FUNCTION_BLOCK FB_ActuatorLinear 

VAR	
	axis: 				AXIS_REF;
	power: 				MC_Power;
	powerOutputs: 		ST_McOutputs;
	moveAbs: 			MC_MoveAbsolute;
	moveAbsOutputs: 	ST_McOutputs;
	reset: 				MC_Reset;
	resetOut: 			ST_McOutputs;
	home:				MC_Home;
	
	
	sID: STRING;
	sDescr: STRING;
	
	
	nLead: UINT := 5;  			// mm per 360deg  - NOT EFFECTIVE YET BECAUSE PITCH IS CURRENTLY HANDLED IN THE AXIS CONFIG
	nStroke: UINT := 100;  		// length of travel
	nHomeOffset: UINT := 0; 	// offset distance from hard-stop for home
	nMaxVel: UINT := 300; 		// mm/s
	nPercentMove: LREAL := 100; 	// % of the full extent of movement (starting from position 0)
	
	eSMState: (INIT, ENABLE, WAIT, FWD_TRIG, FWD, REV_TRIG, REV, ERROR, RESET, HOMING, HOME) := INIT;
	
	fbTONDelay: TON := (PT := T#5S);
	bFirstRun: BOOL := TRUE;
	

	
END_VAR

ActMove();
ActPower();
ActReset();
fbTONDelay();


CASE eSMState OF
	
	INIT:

		IF bFirstRun THEN
			fbTONDelay.IN := TRUE;
			bFirstRun := FALSE;
		END_IF
		
		moveAbs.Execute := FALSE;
		moveAbs.Execute := FALSE;
		reset.Execute := FALSE;
		
		
		IF fbTONDelay.Q THEN
			eSMState := ENABLE;
			fbTONDelay.IN := FALSE;	
			bFirstRun := TRUE;
		END_IF
		
		
		
		
	ENABLE:
	
		IF bFirstRun THEN
			fbTONDelay.IN := TRUE;
			bFirstRun := FALSE;
		END_IF
	
		
		power.Enable := TRUE;
		power.Enable_Positive := TRUE;
		power.Enable_Negative := TRUE;
		
		
		IF power.Status THEN
			eSMState := WAIT;
			fbTONDelay.IN := FALSE;	
			bFirstRun := TRUE;
		(* ELSIF power.Error AND fbTONDelay.Q THEN
			eSMState := ERROR;
			fbTONDelay.IN := FALSE;
			bFirstRun := TRUE; *)
		END_IF
		
	WAIT:
		// Handle eStateTarget command requests here 
		//IF eStateTarget := E_DeviceState.
		
	
	HOMING:
		
		
	FWD_TRIG:
			
			moveAbs.Position := - nStroke * (nPercentMove / 100);		(* mm *)
			moveAbs.Velocity := nMaxVel/2;		(* mm/s *)
			moveAbs.BufferMode := MC_Buffered;  
			moveAbs.Execute := TRUE;
			
			IF moveAbs.Active THEN
				moveAbs.Execute := FALSE;
				fbTONDelay.IN := FALSE;
				eSMState := FWD;
				bFirstRun := TRUE;
			ELSIF moveAbs.CommandAborted OR moveAbs.Error THEN
				eSMState := ERROR;
				bFirstRun := TRUE;
				moveAbs.Execute := FALSE;
			END_IF
				
	FWD:
			eSMState := INIT;
			//eState := FWD;
			
			
			
			
	REV_TRIG:
	
			moveAbs.Position := - (0 + nHomeOffset)  * (nPercentMove / 100);		(* mm *)
			moveAbs.Velocity := nMaxVel/2;										(* mm/s *)
			moveAbs.BufferMode := MC_Buffered;  
			moveAbs.Execute := TRUE;
			
			IF moveAbs.Active THEN
				moveAbs.Execute := FALSE;
				fbTONDelay.IN := FALSE;
				eSMState := REV;
				bFirstRun := TRUE;
			ELSIF moveAbs.CommandAborted OR moveAbs.Error THEN
				eSMState := ERROR;
				bFirstRun := TRUE;
				moveAbs.Execute := FALSE;
			END_IF
			
	REV:
			eSMState := INIT;
			

	ERROR:
			IF axis.Status.Error THEN
				eSMState := RESET;	(* axis error requires reset *)
			ELSE
				eSMState := INIT;		(* function block errors don't need a reset *)
			END_IF
	
	RESET:
	
			IF bFirstRun THEN
				fbTONDelay.IN := TRUE;
				bFirstRun := FALSE;
			END_IF
		
			reset.Execute := TRUE;
			
			IF reset.Done AND fbTONDelay.Q THEN
				eSMState := INIT;
				fbTONDelay.IN := FALSE;
				bFirstRun := TRUE;
			ELSIF reset.Error AND fbTONDelay.Q THEN
				eSMState := ERROR; // the example code pointed this to reset
				fbTONDelay.IN := FALSE;
				bFirstRun := TRUE;
			END_IF
	
	
END_CASE

ACTION ActMove:
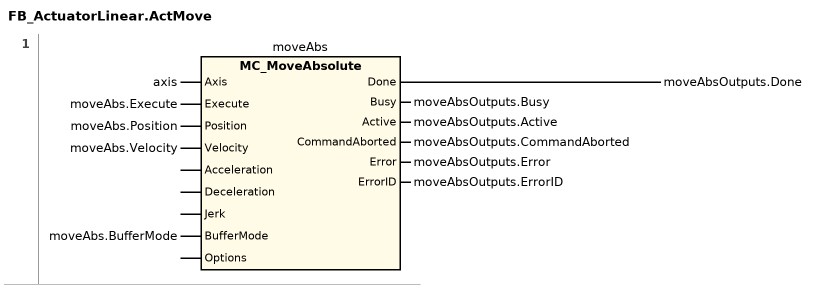
// NETWORK 1
moveAbs(
    Axis := axis,
    Execute := moveAbs.Execute,
    Position := moveAbs.Position,
    Velocity := moveAbs.Velocity,
    BufferMode := moveAbs.BufferMode,
    Busy => moveAbsOutputs.Busy,
    Active => moveAbsOutputs.Active,
    CommandAborted => moveAbsOutputs.CommandAborted,
    Error => moveAbsOutputs.Error,
    ErrorID => moveAbsOutputs.ErrorID); // MC_MoveAbsolute
moveAbsOutputs.Done := moveAbs.Done;
END_ACTION

ACTION ActMove_1:
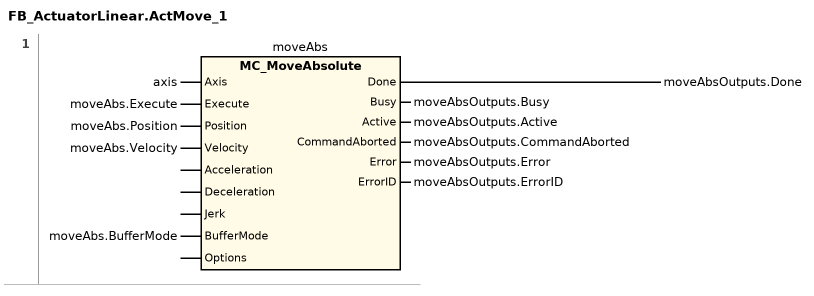
// NETWORK 1
moveAbs(
    Axis := axis,
    Execute := moveAbs.Execute,
    Position := moveAbs.Position,
    Velocity := moveAbs.Velocity,
    BufferMode := moveAbs.BufferMode,
    Busy => moveAbsOutputs.Busy,
    Active => moveAbsOutputs.Active,
    CommandAborted => moveAbsOutputs.CommandAborted,
    Error => moveAbsOutputs.Error,
    ErrorID => moveAbsOutputs.ErrorID); // MC_MoveAbsolute
moveAbsOutputs.Done := moveAbs.Done;
END_ACTION

ACTION ActPower:
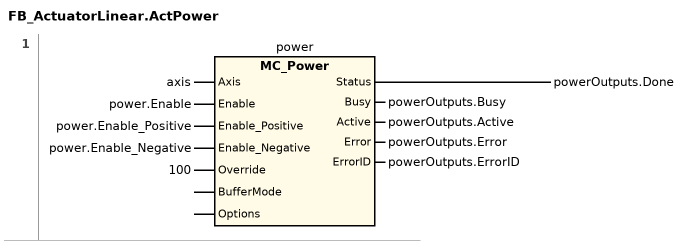
// NETWORK 1
power(
    Axis := axis,
    Enable := power.Enable,
    Enable_Positive := power.Enable_Positive,
    Enable_Negative := power.Enable_Negative,
    Override := 100,
    Busy => powerOutputs.Busy,
    Active => powerOutputs.Active,
    Error => powerOutputs.Error,
    ErrorID => powerOutputs.ErrorID); // MC_Power
powerOutputs.Done := power.Status;
END_ACTION

ACTION ActReset:
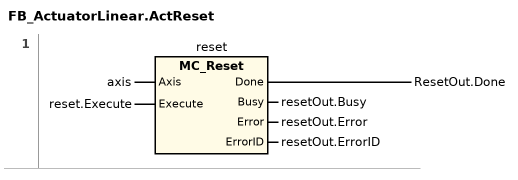
// NETWORK 1
reset(
    Axis := axis,
    Execute := reset.Execute,
    Busy => resetOut.Busy,
    Error => resetOut.Error,
    ErrorID => resetOut.ErrorID); // MC_Reset
ResetOut.Done := reset.Done;
END_ACTION

METHOD extend : BOOL
VAR_INPUT
END_VAR
IF eSMState = WAIT THEN
	eSMState := FWD_TRIG;
	nPercentMove := 100;
	extend := TRUE;
ELSE
	extend := FALSE;
END_IF
END_METHOD

METHOD FB_init : BOOL
VAR_INPUT
	bInitRetains : BOOL; // if TRUE, the retain variables are initialized (warm start / cold start)
	bInCopyCode : BOOL;  // if TRUE, the instance afterwards gets moved into the copy code (online change)
	
	ID: STRING;
	Descr: STRING;
	
	Lead: UINT;  			// mm per 360deg
	Stroke: UINT;  		// length of travel
	HomeOffset: UINT; 	// offset distance from hard-stop for home
END_VAR

sID := ID;
sDescr := Descr;

nLead := Lead;
nStroke := Stroke;
nHomeOffset := HomeOffset;
END_METHOD

METHOD initialise : BOOL
VAR_INPUT
	
	Lead: UINT;  			// mm per 360deg
	Stroke: UINT;  		// length of travel
	HomeOffset: UINT; 	// offset distance from hard-stop for home
END_VAR
nLead := Lead;
nStroke := Stroke;
nHomeOffset := HomeOffset;
END_METHOD

METHOD moveToPos : BOOL
VAR_INPUT
	PercStroke: LREAL;
END_VAR
IF eSMState = WAIT THEN
	eSMState := FWD_TRIG;
	nPercentMove := PercStroke;
	moveToPos := TRUE;
ELSE
	moveToPos := FALSE;
END_IF
END_METHOD

METHOD retract : BOOL
VAR_INPUT
END_VAR
IF eSMState = WAIT THEN
	eSMState := REV_TRIG;
	nPercentMove := 100;
	retract := TRUE;
ELSE
	retract := FALSE;
END_IF
END_METHOD

END_FUNCTION_BLOCK

(* stored: Version 1.1.0.1, ProductVersion 3.1.4024.12
   POU FB_ActuatorLinear: Id {c97eae7a-0e8d-4184-b960-b43b650074d1}, SpecialFunc None
   Action ActMove: Id {7f77cf4e-6c43-4127-a3d4-65c05e838a38}
   Action ActMove_1: Id {2ea978d5-2b0d-40d2-875e-63da86789a91}
   Action ActPower: Id {6246be74-b5bf-45a6-9e07-4b93eadeb7de}
   Action ActReset: Id {d97ef662-b6e5-4f0b-8a6c-ca88ac7e4163}
   Method extend: Id {97662ec9-efbc-4a54-a824-cc13520cf22d}
   Method FB_init: Id {4e129cbb-940c-4f3b-8804-40d3aa72d4e6}
   Method initialise: Id {8d611d04-ba4f-4e5b-9758-13d91fb52e52}
   Method moveToPos: Id {d155c808-00e7-45f5-9930-b1d3bfe5fd56}
   Method retract: Id {d8fa0476-ce8c-4bc5-b226-abc1a4d045c9} *)
